// TIA Portal project "Projekt Inżynierski" (V15.1)

(* hardware
DEVICE "S7-1200 station_1"  S7-1200 Station
   slot 0: "Rack_0"  S7-1200 Rack  Rack  V1.0
   slot 1: "PLC_1"  CPU 1214C DC/DC/DC  6ES7 214-1AG40-0XB0  V4.1
      slot 3: "AQ 1x12BIT_1"  AQ1 signal board  6ES7 232-4HA30-0XB0  V1.0
*)

// ===== PLC "PLC_1"  CPU 1214C DC/DC/DC =====

VAR_GLOBAL   // PLC tag table "Default tag table"
   "Tag_1" AT %IW64 : Word;
   "Tag_2" AT %MD10 : Real;
   "Engine Power Suply" AT %MW50 : Int;
   "Tag_4" AT %IW66 : Int;
   "Tag_5" AT %MD11 : Real;
   "Tag_6" AT %MD12 : Real;
   "Tag_7" AT %MD13 : Real;
   "Lindar Power Suply" AT %MW51 : Int;
   "WiFi Power Suply" AT %MW52 : Int;
   "Tag_10" AT %MD14 : Real;
   "Tag_11" AT %MD15 : Real;
   "Battery Voltage Output" AT %MW2 : Int;
   "Tag_3" AT %MD17 : Real;
   "Tag_8" AT %MD18 : Real;
   "Battery Power Suply" AT %MW53 : Int;
   "System_Byte" AT %MB1 : Byte;
   "FirstScan" AT %M1.0 : Bool;
   "DiagStatusUpdate" AT %M1.1 : Bool;
   "AlwaysTRUE" AT %M1.2 : Bool;
   "AlwaysFALSE" AT %M1.3 : Bool;
   "Clock_Byte" AT %MB0 : Byte;
   "Clock_10Hz" AT %M0.0 : Bool;
   "Clock_5Hz" AT %M0.1 : Bool;
   "Clock_2.5Hz" AT %M0.2 : Bool;
   "Clock_2Hz" AT %M0.3 : Bool;
   "Clock_1.25Hz" AT %M0.4 : Bool;
   "Clock_1Hz" AT %M0.5 : Bool;
   "Clock_0.625Hz" AT %M0.6 : Bool;
   "Clock_0.5Hz" AT %M0.7 : Bool;
   "Tag_9" AT %MD19 : Real;
   "Tag_12" AT %MD20 : Real;
   "Tag_13" AT %MD21 : DWord;
   "Tag_14" AT %Q1.0 : Bool;
   "Tag_15" AT %MD22 : DWord;
   "Tag_16" AT %MW54 : Int;   // New Engine Power Suply
   "Tag_17" AT %MW56 : Int;   // New Lidar Power Suply
   "Tag_18" AT %MW58 : Int;   // New Wifi Power Suply
   "Tag_19" AT %MW60 : Int;
   "Tag_20" AT %Q1.1 : Bool;
   "Tag_21" AT %MW70 : Int;
   "Tag_22" AT %MW72 : Int;
   "Tag_23" AT %MW74 : Int;
   "Tag_24" AT %MW76 : Int;
   "Tag_25" AT %MW80 : Int;
   "Tag_26" AT %Q1.2 : Bool;
   "Tag_27" AT %Q1.3 : Bool;
   "Tag_28" AT %MW90 : Int;
   "Tag_29" AT %MW91 : Int;
   "Tag_30" AT %MW92 : Int;
   "Tag_31" AT %MW93 : Int;
   "Tag_32" AT %MW94 : Int;
   "Tag_33" AT %MW95 : Int;
   "Tag_34" AT %Q1.4 : Bool;
   "Tag_35" AT %Q1.5 : Bool;
   "Tag_36" AT %MW96 : Int;
   "Tag_37" AT %MW97 : Int;
   "Tag_38" AT %MW98 : Int;
   "Tag_39" AT %MW30 : Int;
   "Tag_40" AT %MW32 : Int;
   "Tag_41" AT %MW34 : Int;
   "Tag_42" AT %MW35 : Int;
   "Tag_43" AT %MW40 : Int;
   "Tag_44" AT %MW42 : Int;
   "Tag_45" AT %MW44 : Int;
   "Tag_46" AT %Q1.6 : Bool;
   "Tag_47" AT %Q1.7 : Bool;
   "Tag_48" AT %MD24 : Time;
   "Tag_49" AT %Q2.1 : Bool;
END_VAR

DATA_BLOCK "Agregation of Current data"   // DB1
{ S7_Optimized_Access := 'TRUE' }
VERSION : 0.1
   VAR
      "Engine Current" : Int;
      "Wi-Fi Current" : Int;
      "Power Source current" : Int;
      "Lidar Current" : Int;
      "Battery Voltage" : Int;
      "Engine Power Useage" : Int;
      "Lidar Power Useage" : Int;
      "Wi-Fi Power Useage" : Int;
      "Battery Power Useage" : Int;
      "Momental Power Useage" : Int;
      "Energy useage" : Int;
   END_VAR
BEGIN
END_DATA_BLOCK

DATA_BLOCK "TCPIP_COMMUNICATION_DB"   // DB2
{ S7_Optimized_Access := 'TRUE' }
VERSION : 0.1
BEGIN
END_DATA_BLOCK

DATA_BLOCK "DATA_TO_SEND"   // DB7
{ S7_Optimized_Access := 'TRUE' }
VERSION : 0.1
   VAR
      RECIVE : Array[0..20] of Char;
      SEND : Array[0..7] of Int;
   END_VAR
BEGIN
END_DATA_BLOCK

DATA_BLOCK "TCPIP_COMMUNICATION_DB_1"   // DB9
{ S7_Optimized_Access := 'TRUE' }
VERSION : 0.1
// stored: InstanceOfName TCPIP_COMMUNICATION
"TCPIP_COMMUNICATION"
BEGIN
END_DATA_BLOCK

DATA_BLOCK "Integration Testing DataBase"   // DB12
{ S7_Optimized_Access := 'TRUE' }
VERSION : 0.1
   VAR
      "1HZ" : Int;
      "0.5HZ" : Int;
      "1.25HZ" : Int;
      "2HZ" : Int;
      "2.5HZ" : Int;
      "0.625" : Int;
   END_VAR
BEGIN
END_DATA_BLOCK

// folder: System blocks/Program resources

DATA_BLOCK "IEC_Counter_0_DB_1"   // DB4
{ S7_Optimized_Access := 'TRUE' }
AUTHOR : Simatic
FAMILY : IEC
NAME : CNTR
VERSION : 1.0
// stored: InstanceOfName IEC_COUNTER
"IEC_COUNTER"
BEGIN
END_DATA_BLOCK

DATA_BLOCK "IEC_Counter_0_DB"   // DB10
{ S7_Optimized_Access := 'TRUE' }
AUTHOR : Simatic
FAMILY : IEC
NAME : CNTR
VERSION : 1.0
// stored: InstanceOfName IEC_COUNTER
"IEC_COUNTER"
BEGIN
END_DATA_BLOCK

DATA_BLOCK "IEC_Counter_0_DB_2"   // DB11
{ S7_Optimized_Access := 'TRUE' }
AUTHOR : Simatic
FAMILY : IEC
NAME : CNTR
VERSION : 1.0
// stored: InstanceOfName IEC_COUNTER
"IEC_COUNTER"
BEGIN
END_DATA_BLOCK

DATA_BLOCK "IEC_Timer_0_DB"   // DB18
{ S7_Optimized_Access := 'TRUE' }
AUTHOR : Simatic
FAMILY : IEC
NAME : IEC_TMR
VERSION : 1.0
// stored: InstanceOfName IEC_TIMER
"IEC_TIMER"
BEGIN
END_DATA_BLOCK

DATA_BLOCK "IEC_Timer_0_DB_1"   // DB19
{ S7_Optimized_Access := 'TRUE' }
AUTHOR : Simatic
FAMILY : IEC
NAME : IEC_TMR
VERSION : 1.0
// stored: InstanceOfName IEC_TIMER
"IEC_TIMER"
BEGIN
END_DATA_BLOCK

DATA_BLOCK "IEC_Timer_0_DB_2"   // DB20
{ S7_Optimized_Access := 'TRUE' }
AUTHOR : Simatic
FAMILY : IEC
NAME : IEC_TMR
VERSION : 1.0
// stored: InstanceOfName IEC_TIMER
"IEC_TIMER"
BEGIN
END_DATA_BLOCK

DATA_BLOCK "IEC_Timer_0_DB_3"   // DB21
{ S7_Optimized_Access := 'TRUE' }
AUTHOR : Simatic
FAMILY : IEC
NAME : IEC_TMR
VERSION : 1.0
// stored: InstanceOfName IEC_TIMER
"IEC_TIMER"
BEGIN
END_DATA_BLOCK

DATA_BLOCK "IEC_Counter_0_DB_3"   // DB22
{ S7_Optimized_Access := 'TRUE' }
AUTHOR : Simatic
FAMILY : IEC
NAME : CNTR
VERSION : 1.0
// stored: InstanceOfName IEC_COUNTER
"IEC_COUNTER"
BEGIN
END_DATA_BLOCK

// folder: (top level)

FUNCTION_BLOCK "TCPIP_COMMUNICATION"   // FB1, LAD
{ S7_Optimized_Access := 'TRUE' }
VERSION : 0.1
   VAR
      TCON : Struct
         REQ : Bool;
         DONE : Bool := false;
         BUSY : Bool;
         ERROR : Bool;
         STATUS : UInt;
         DONESAVE : Bool;
         CONNECT : UInt;
      END_STRUCT;
      TDCON : Struct
         REQ : Bool;
         DONE : Bool;
         BUSY : Bool;
         ERROR : Bool;
         STATUS : UInt;
      END_STRUCT;
      TSEND : Struct
         REQ : Bool;
         DONE : Bool;
         BUSY : Bool;
         ERROR : Bool;
         STATUS : UInt;
      END_STRUCT;
      TRECIVE : Struct
         EN_R : Bool;
         NDR : Bool;
         BUSY : Bool;
         ERROR : Bool;
         STATUS : UInt;
         RCVD_LEN : UInt;
      END_STRUCT;
   END_VAR
BEGIN

REGION Network 1: TCON
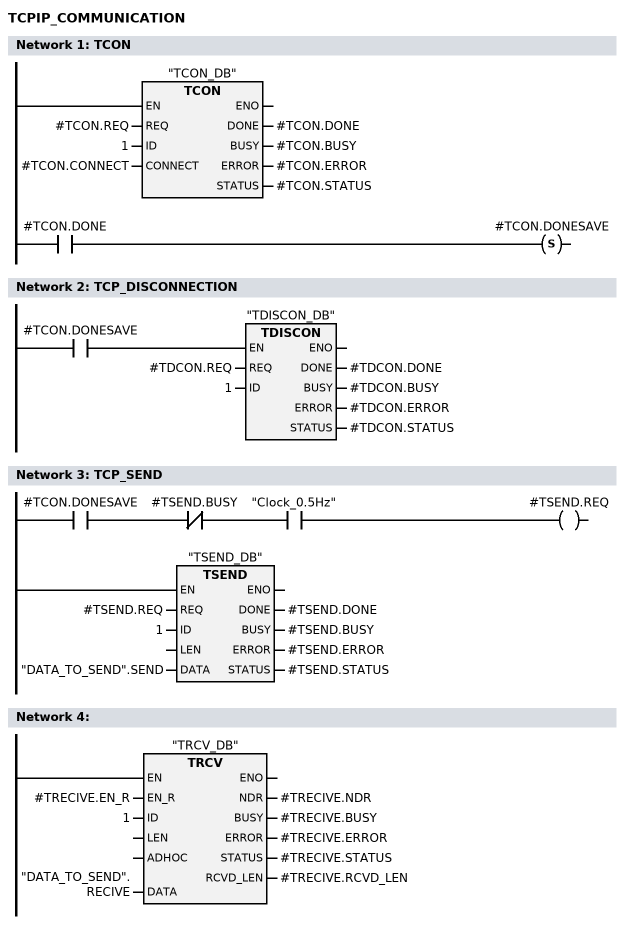
   "TCON_DB"(REQ := #TCON.REQ,   // TCON
             ID := 1,
             CONNECT := #TCON.CONNECT,
             DONE => #TCON.DONE,
             BUSY => #TCON.BUSY,
             ERROR => #TCON.ERROR,
             STATUS => #TCON.STATUS);
   IF #TCON.DONE THEN #TCON.DONESAVE := TRUE; END_IF;
END_REGION

REGION Network 2: TCP_DISCONNECTION
   IF #TCON.DONESAVE THEN
       "TDISCON_DB"(REQ := #TDCON.REQ,   // TDISCON
                    ID := 1,
                    DONE => #TDCON.DONE,
                    BUSY => #TDCON.BUSY,
                    ERROR => #TDCON.ERROR,
                    STATUS => #TDCON.STATUS);
   END_IF;
END_REGION

REGION Network 3: TCP_SEND
   #TSEND.REQ := #TCON.DONESAVE AND NOT #TSEND.BUSY AND "Clock_0.5Hz";
   "TSEND_DB"(REQ := #TSEND.REQ,   // TSEND
              ID := 1,
              DATA := "DATA_TO_SEND".SEND,
              DONE => #TSEND.DONE,
              BUSY => #TSEND.BUSY,
              ERROR => #TSEND.ERROR,
              STATUS => #TSEND.STATUS);
END_REGION

REGION Network 4
   "TRCV_DB"(EN_R := #TRECIVE.EN_R,   // TRCV
             ID := 1,
             DATA := "DATA_TO_SEND".RECIVE,
             NDR => #TRECIVE.NDR,
             BUSY => #TRECIVE.BUSY,
             ERROR => #TRECIVE.ERROR,
             STATUS => #TRECIVE.STATUS,
             RCVD_LEN => #TRECIVE.RCVD_LEN);
END_REGION
END_FUNCTION_BLOCK

FUNCTION "Block_1" : Void   // FC1, LAD
{ S7_Optimized_Access := 'TRUE' }
VERSION : 0.1
   VAR_INPUT
      "%IW64" : Array[0..1] of Byte;
   END_VAR
BEGIN
END_FUNCTION

ORGANIZATION_BLOCK "Main"   // OB1, LAD, ProgramCycle
TITLE = "Main Program Sweep (Cycle)"
{ S7_Optimized_Access := 'TRUE' }
VERSION : 0.1
   VAR_INPUT
      Initial_Call : Bool;   // Initial call of this OB
      Remanence : Bool;   // =True, if remanent data are available
   END_VAR
   VAR_TEMP
      Clk_output : Bool;
   END_VAR
BEGIN

REGION Network 1: Get Engine Power Suply
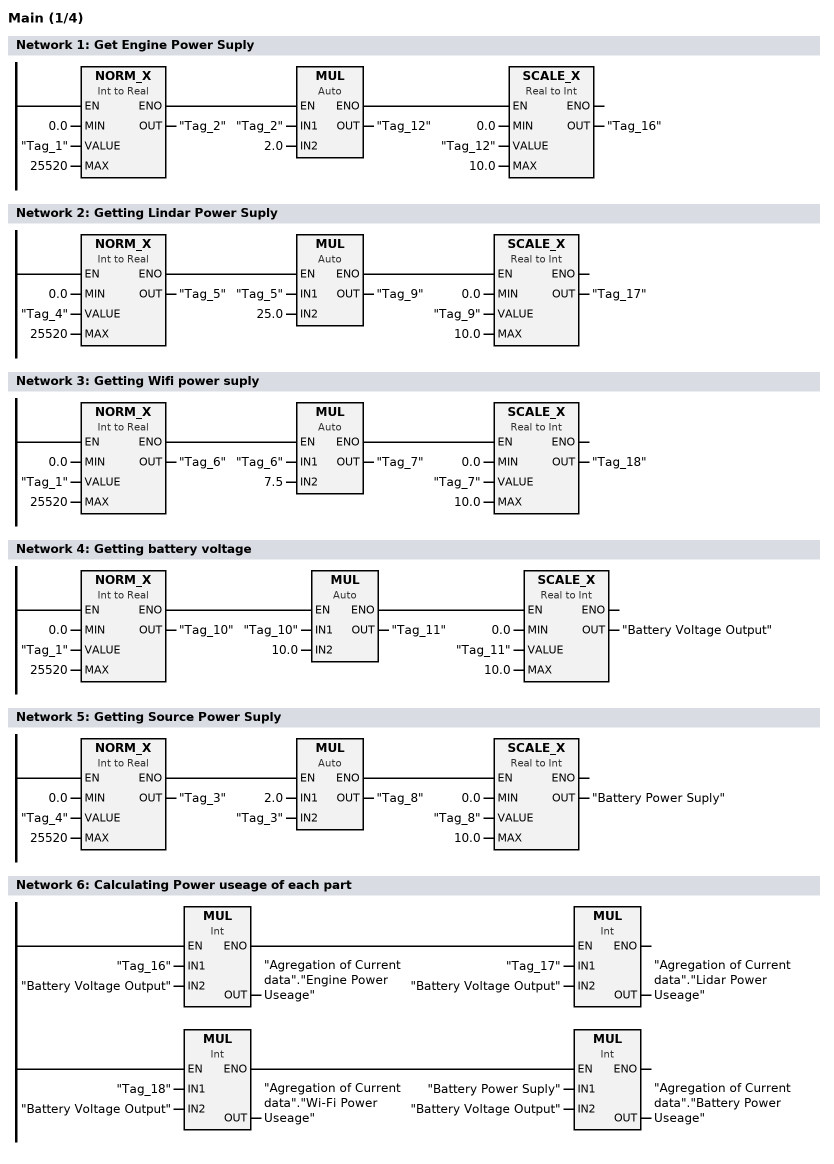
   RUNG wire#powerrail
      { S7_Templates := "[SrcType := Int, DestType := Real]" } Normalize(min := 0.0, value := "Tag_1", max := 25520, out => "Tag_2")
      Mul(in1 := "Tag_2", in2 := 2.0, out => "Tag_12")
      { S7_Templates := "[SrcType := Real, DestType := Int]" } Scale(min := 0.0, value := "Tag_12", max := 10.0, out => "Tag_16")
   END_RUNG
   // the same network as SCL:
   "Tag_2" := NORM_X(MIN := 0.0, VALUE := "Tag_1", MAX := 25520);
   "Tag_12" := "Tag_2" * 2.0;
   "Tag_16" := SCALE_X(MIN := 0.0, VALUE := "Tag_12", MAX := 10.0);
END_REGION

REGION Network 2: Getting Lindar Power Suply
   RUNG wire#powerrail
      { S7_Templates := "[SrcType := Int, DestType := Real]" } Normalize(min := 0.0, value := "Tag_4", max := 25520, out => "Tag_5")
      Mul(in1 := "Tag_5", in2 := 25.0, out => "Tag_9")
      { S7_Templates := "[SrcType := Real, DestType := Int]" } Scale(min := 0.0, value := "Tag_9", max := 10.0, out => "Tag_17")
   END_RUNG
   // the same network as SCL:
   "Tag_5" := NORM_X(MIN := 0.0, VALUE := "Tag_4", MAX := 25520);
   "Tag_9" := "Tag_5" * 25.0;
   "Tag_17" := SCALE_X(MIN := 0.0, VALUE := "Tag_9", MAX := 10.0);
END_REGION

REGION Network 3: Getting Wifi power suply
   RUNG wire#powerrail
      { S7_Templates := "[SrcType := Int, DestType := Real]" } Normalize(min := 0.0, value := "Tag_1", max := 25520, out => "Tag_6")
      Mul(in1 := "Tag_6", in2 := 7.5, out => "Tag_7")
      { S7_Templates := "[SrcType := Real, DestType := Int]" } Scale(min := 0.0, value := "Tag_7", max := 10.0, out => "Tag_18")
   END_RUNG
   // the same network as SCL:
   "Tag_6" := NORM_X(MIN := 0.0, VALUE := "Tag_1", MAX := 25520);
   "Tag_7" := "Tag_6" * 7.5;
   "Tag_18" := SCALE_X(MIN := 0.0, VALUE := "Tag_7", MAX := 10.0);
END_REGION

REGION Network 4: Getting battery voltage
   RUNG wire#powerrail
      { S7_Templates := "[SrcType := Int, DestType := Real]" } Normalize(min := 0.0, value := "Tag_1", max := 25520, out => "Tag_10")
      Mul(in1 := "Tag_10", in2 := 10.0, out => "Tag_11")
      { S7_Templates := "[SrcType := Real, DestType := Int]" } Scale(min := 0.0, value := "Tag_11", max := 10.0, out => "Battery Voltage Output")
   END_RUNG
   // the same network as SCL:
   "Tag_10" := NORM_X(MIN := 0.0, VALUE := "Tag_1", MAX := 25520);
   "Tag_11" := "Tag_10" * 10.0;
   "Battery Voltage Output" := SCALE_X(MIN := 0.0, VALUE := "Tag_11", MAX := 10.0);
END_REGION

REGION Network 5: Getting Source Power Suply
   RUNG wire#powerrail
      { S7_Templates := "[SrcType := Int, DestType := Real]" } Normalize(min := 0.0, value := "Tag_4", max := 25520, out => "Tag_3")
      Mul(in1 := 2.0, in2 := "Tag_3", out => "Tag_8")
      { S7_Templates := "[SrcType := Real, DestType := Int]" } Scale(min := 0.0, value := "Tag_8", max := 10.0, out => "Battery Power Suply")
   END_RUNG
   // the same network as SCL:
   "Tag_3" := NORM_X(MIN := 0.0, VALUE := "Tag_4", MAX := 25520);
   "Tag_8" := 2.0 * "Tag_3";
   "Battery Power Suply" := SCALE_X(MIN := 0.0, VALUE := "Tag_8", MAX := 10.0);
END_REGION

REGION Network 6: Calculating Power useage of each part
   RUNG wire#powerrail
      { S7_Templates := "SrcType := Int" } Mul(in1 := "Tag_16", in2 := "Battery Voltage Output", out => "Agregation of Current data"."Engine Power Useage")
      { S7_Templates := "SrcType := Int" } Mul(in1 := "Tag_17", in2 := "Battery Voltage Output", out => "Agregation of Current data"."Lidar Power Useage")
   END_RUNG
   RUNG wire#powerrail
      { S7_Templates := "SrcType := Int" } Mul(in1 := "Tag_18", in2 := "Battery Voltage Output", out => "Agregation of Current data"."Wi-Fi Power Useage")
      { S7_Templates := "SrcType := Int" } Mul(in1 := "Battery Power Suply", in2 := "Battery Voltage Output", out => "Agregation of Current data"."Battery Power Useage")
   END_RUNG
   // the same network as SCL:
   "Agregation of Current data"."Engine Power Useage" := "Tag_16" * "Battery Voltage Output";
   "Agregation of Current data"."Lidar Power Useage" := "Tag_17" * "Battery Voltage Output";
   "Agregation of Current data"."Wi-Fi Power Useage" := "Tag_18" * "Battery Voltage Output";
   "Agregation of Current data"."Battery Power Useage" := "Battery Power Suply" * "Battery Voltage Output";
END_REGION

REGION Network 7: Calculating Total Energy Consumption
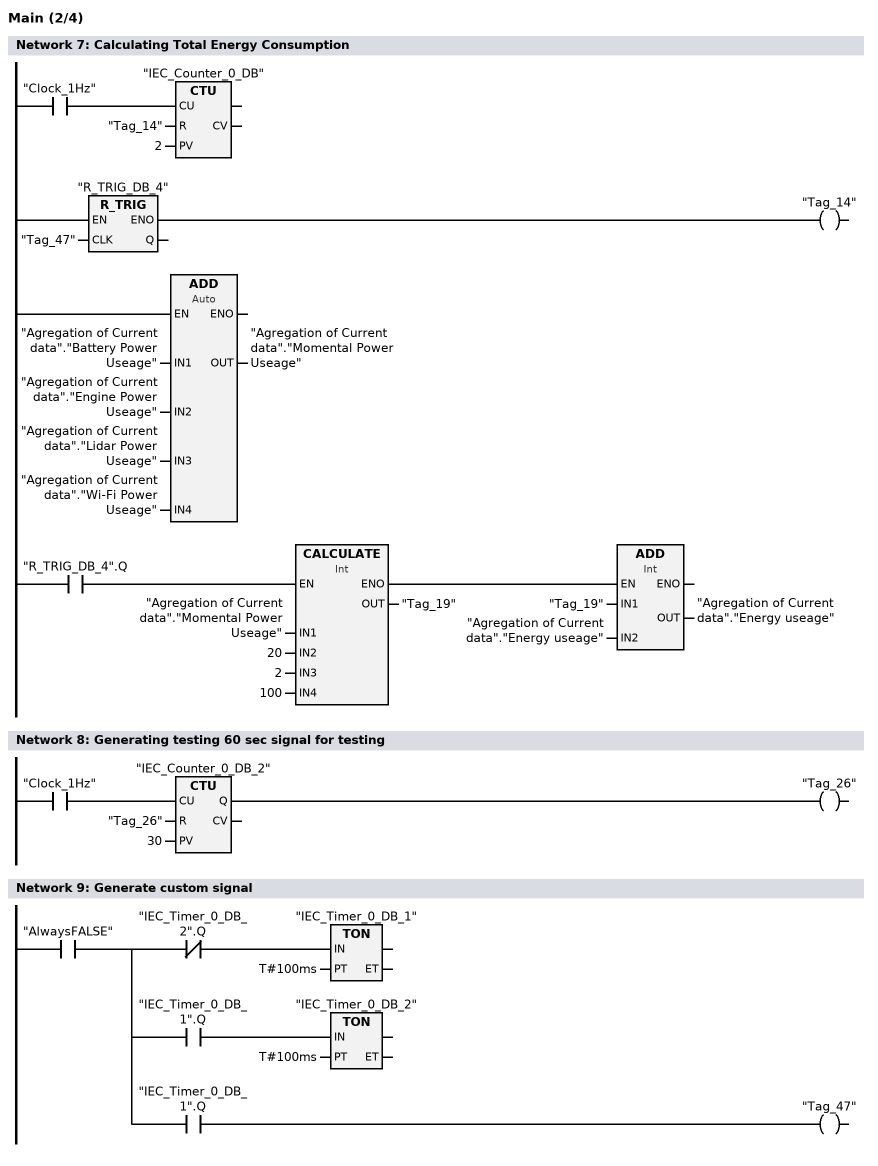
   // ENO of a box is taken as its EN; it also drops when the box reports an error
   "IEC_Counter_0_DB".CTU(CU := "Clock_1Hz", R := "Tag_14", PV := 2);
   "R_TRIG_DB_4"(CLK := "Tag_47");   // R_TRIG
   "Tag_14" := TRUE;
   "Agregation of Current data"."Momental Power Useage" := "Agregation of Current data"."Battery Power Useage" + "Agregation of Current data"."Engine Power Useage" + "Agregation of Current data"."Lidar Power Useage" + "Agregation of Current data"."Wi-Fi Power Useage";
   IF "R_TRIG_DB_4".Q THEN
       "Tag_19" := "Agregation of Current data"."Momental Power Useage"*20/(2*100);
       "Agregation of Current data"."Energy useage" := "Tag_19" + "Agregation of Current data"."Energy useage";
   END_IF;
END_REGION

REGION Network 8: Generating testing 60 sec signal for testing
   "IEC_Counter_0_DB_2".CTU(CU := "Clock_1Hz", R := "Tag_26", PV := 30);
   "Tag_26" := "IEC_Counter_0_DB_2".Q;
END_REGION

REGION Network 9: Generate custom signal
   "IEC_Timer_0_DB_1".TON(IN := "AlwaysFALSE" AND NOT "IEC_Timer_0_DB_2".Q, PT := T#100ms);
   "IEC_Timer_0_DB_2".TON(IN := "AlwaysFALSE" AND "IEC_Timer_0_DB_1".Q, PT := T#100ms);
   "Tag_47" := "AlwaysFALSE" AND "IEC_Timer_0_DB_1".Q;
END_REGION

REGION Network 10
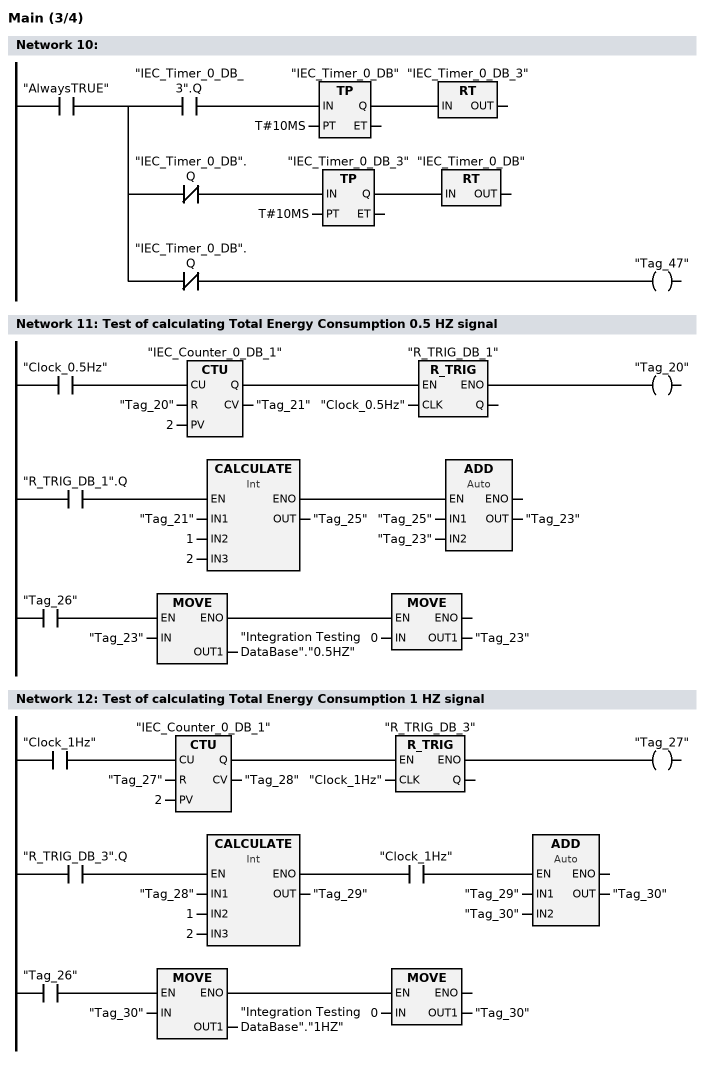
   "IEC_Timer_0_DB".TP(IN := "AlwaysTRUE" AND "IEC_Timer_0_DB_3".Q, PT := T#10MS);
   IF "IEC_Timer_0_DB".Q THEN RESET_TIMER("IEC_Timer_0_DB_3"); END_IF;
   "IEC_Timer_0_DB_3".TP(IN := "AlwaysTRUE" AND NOT "IEC_Timer_0_DB".Q, PT := T#10MS);
   IF "IEC_Timer_0_DB_3".Q THEN RESET_TIMER("IEC_Timer_0_DB"); END_IF;
   "Tag_47" := "AlwaysTRUE" AND NOT "IEC_Timer_0_DB".Q;
END_REGION

REGION Network 11: Test of calculating Total Energy Consumption 0.5 HZ signal
   // ENO of a box is taken as its EN; it also drops when the box reports an error
   "IEC_Counter_0_DB_1".CTU(CU := "Clock_0.5Hz", R := "Tag_20", PV := 2, CV => "Tag_21");
   IF "IEC_Counter_0_DB_1".Q THEN
       "R_TRIG_DB_1"(CLK := "Clock_0.5Hz");   // R_TRIG
   END_IF;
   "Tag_20" := "IEC_Counter_0_DB_1".Q;
   IF "R_TRIG_DB_1".Q THEN
       "Tag_25" := "Tag_21"*1/2;
       "Tag_23" := "Tag_25" + "Tag_23";
   END_IF;
   IF "Tag_26" THEN
       "Integration Testing DataBase"."0.5HZ" := "Tag_23";
       "Tag_23" := 0;
   END_IF;
END_REGION

REGION Network 12: Test of calculating Total Energy Consumption 1 HZ signal
   // ENO of a box is taken as its EN; it also drops when the box reports an error
   "IEC_Counter_0_DB_1".CTU(CU := "Clock_1Hz", R := "Tag_27", PV := 2, CV => "Tag_28");
   IF "IEC_Counter_0_DB_1".Q THEN
       "R_TRIG_DB_3"(CLK := "Clock_1Hz");   // R_TRIG
   END_IF;
   "Tag_27" := "IEC_Counter_0_DB_1".Q;
   IF "R_TRIG_DB_3".Q THEN "Tag_29" := "Tag_28"*1/2; END_IF;
   IF "R_TRIG_DB_3".Q AND "Clock_1Hz" THEN "Tag_30" := "Tag_29" + "Tag_30"; END_IF;
   IF "Tag_26" THEN
       "Integration Testing DataBase"."1HZ" := "Tag_30";
       "Tag_30" := 0;
   END_IF;
END_REGION

REGION Network 13: Testing clock 0.625
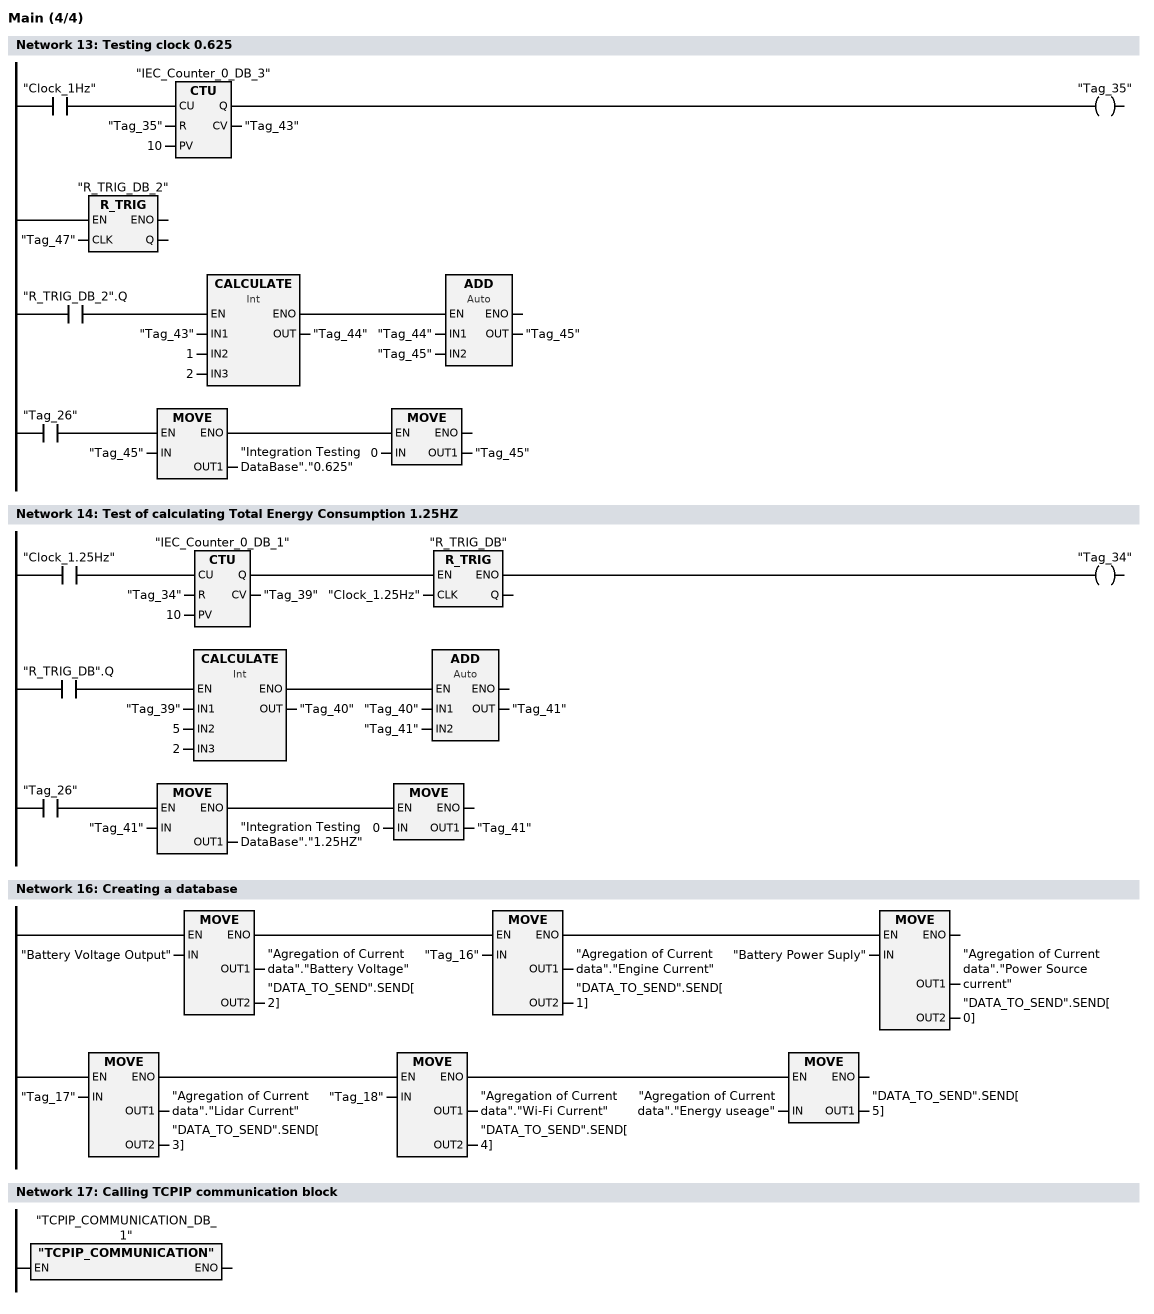
   "IEC_Counter_0_DB_3".CTU(CU := "Clock_1Hz", R := "Tag_35", PV := 10, CV => "Tag_43");
   "Tag_35" := "IEC_Counter_0_DB_3".Q;
   "R_TRIG_DB_2"(CLK := "Tag_47");   // R_TRIG
   IF "R_TRIG_DB_2".Q THEN
       "Tag_44" := "Tag_43"*1/2;
       "Tag_45" := "Tag_44" + "Tag_45";
   END_IF;
   IF "Tag_26" THEN
       "Integration Testing DataBase"."0.625" := "Tag_45";
       "Tag_45" := 0;
   END_IF;
END_REGION

REGION Network 14: Test of calculating Total Energy Consumption 1.25HZ
   // ENO of a box is taken as its EN; it also drops when the box reports an error
   "IEC_Counter_0_DB_1".CTU(CU := "Clock_1.25Hz", R := "Tag_34", PV := 10, CV => "Tag_39");
   IF "IEC_Counter_0_DB_1".Q THEN
       "R_TRIG_DB"(CLK := "Clock_1.25Hz");   // R_TRIG
   END_IF;
   "Tag_34" := "IEC_Counter_0_DB_1".Q;
   IF "R_TRIG_DB".Q THEN
       "Tag_40" := "Tag_39"*5/2;
       "Tag_41" := "Tag_40" + "Tag_41";
   END_IF;
   IF "Tag_26" THEN
       "Integration Testing DataBase"."1.25HZ" := "Tag_41";
       "Tag_41" := 0;
   END_IF;
END_REGION

REGION Network 16: Creating a database
   RUNG wire#powerrail
      Move(in := "Battery Voltage Output", out1 => "Agregation of Current data"."Battery Voltage", out2 => "DATA_TO_SEND".SEND[2])
      Move(in := "Tag_16", out1 => "Agregation of Current data"."Engine Current", out2 => "DATA_TO_SEND".SEND[1])
      Move(in := "Battery Power Suply", out1 => "Agregation of Current data"."Power Source current", out2 => "DATA_TO_SEND".SEND[0])
   END_RUNG
   RUNG wire#powerrail
      Move(in := "Tag_17", out1 => "Agregation of Current data"."Lidar Current", out2 => "DATA_TO_SEND".SEND[3])
      Move(in := "Tag_18", out1 => "Agregation of Current data"."Wi-Fi Current", out2 => "DATA_TO_SEND".SEND[4])
      Move(in := "Agregation of Current data"."Energy useage", out1 => "DATA_TO_SEND".SEND[5])
   END_RUNG
   // the same network as SCL:
   "Agregation of Current data"."Battery Voltage" := "Battery Voltage Output";
   "DATA_TO_SEND".SEND[2] := "Battery Voltage Output";
   "Agregation of Current data"."Engine Current" := "Tag_16";
   "DATA_TO_SEND".SEND[1] := "Tag_16";
   "Agregation of Current data"."Power Source current" := "Battery Power Suply";
   "DATA_TO_SEND".SEND[0] := "Battery Power Suply";
   "Agregation of Current data"."Lidar Current" := "Tag_17";
   "DATA_TO_SEND".SEND[3] := "Tag_17";
   "Agregation of Current data"."Wi-Fi Current" := "Tag_18";
   "DATA_TO_SEND".SEND[4] := "Tag_18";
   "DATA_TO_SEND".SEND[5] := "Agregation of Current data"."Energy useage";
END_REGION

REGION Network 17: Calling TCPIP communication block
   RUNG wire#powerrail
      "TCPIP_COMMUNICATION_DB_1"()
   END_RUNG
   // the same network as SCL:
   "TCPIP_COMMUNICATION_DB_1"();   // "TCPIP_COMMUNICATION"
END_REGION
END_ORGANIZATION_BLOCK